RESOURCE_TYPE PANEL_RESOURCE (* Resource for graphic Panel *)
  (* Standard: 61499-2 *)
  (* Version 0.2, 2000-05-28, JHC, Rockwell Automation, Set E_RESTART position. *)
  (* Version 0.1, 2000-05-10, JHC, Rockwell Automation, Removed "Speed" Attribute *)
  (* Version 0.0, 2000-01-25, JHC, Rockwell Automation, Testing "Speed" Attribute *)
  (* Compiler header: package fb.rt.jfc; import java.awt.*; *)
  (* Compiler Java IBM VisualAge 3.0 *)
  VAR_INPUT
    TRACE : BOOL; (* True=trace enabled,default is false *)
    ROWS : DINT; (* Rows(if any)in grid layout *)
    COLS : DINT; (* Columns(if any)in grid layout *)
  END_VAR
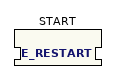
  FBS
    START : E_RESTART;
  END_FBS
END_RESOURCE_TYPE
